// TIA Portal project "P10" (V20)

(* hardware
DEVICE "S7-1200 station_1"  S7-1200 Station
   slot 0: "Rack_0"  S7-1200 Rack  Rack  V1.0
   slot 1: "PLC_1"  CPU 1214C DC/DC/DC  6ES7 214-1AG40-0XB0  V4.7
*)

// ===== PLC "PLC_1"  CPU 1214C DC/DC/DC =====

VAR_GLOBAL   // PLC tag table "Default tag table"
   "IN" AT %M0.0 : Bool;
   "O_TP" AT %M0.1 : Bool;
   "To_TP" AT %MD2 : Time;
   "To_TON" AT %MD6 : Time;
   "O_TON" AT %M0.2 : Bool;
   "To_TOF" AT %MD10 : Time;
   "O_TOF" AT %M0.3 : Bool;
   "Reset" AT %M0.5 : Bool;
   "To_TONR" AT %MD14 : Time;
   "O_TONR" AT %M0.4 : Bool;
   "OCOUNT_CTU" AT %MW18 : Int;
   "Q_CTU" AT %M0.6 : Bool;
   "cargar" AT %M0.7 : Bool;
   "OCOUNT_CTD" AT %MW20 : Int;
   "Q_CTD" AT %M1.0 : Bool;
   "Incremento" AT %M1.1 : Bool;
   "Decremento" AT %M1.2 : Bool;
   "QD_CTUD_Menor0" AT %M1.3 : Bool;
   "conteo" AT %MW22 : Int;
   "QU_CTUD_MAYOR_PV" AT %M1.4 : Bool;
   "enclavamiento" AT %M2.0 : Bool;
   "Verde" AT %Q0.0 : Bool;
   "Tag_3" AT %MD18 : Time;
   "parada" AT %I0.1 : Bool;
   "Amarillo" AT %Q0.1 : Bool;
   "Rojo" AT %Q0.2 : Bool;
   "5srojo" AT %M2.5 : Bool;
   "Tag_2" AT %I0.2 : Bool;
   "Tag_4" AT %M2.2 : Bool;
   "Contador" AT %M2.3 : Bool;
   "reset_cont_sem" AT %M2.4 : Bool;
END_VAR

// folder: System blocks/Program resources

DATA_BLOCK "IEC_Timer_0_DB_5"   // DB8
{ S7_Optimized_Access := 'TRUE' }
AUTHOR : Simatic
FAMILY : IEC
NAME : IEC_TMR
VERSION : 1.0
// stored: InstanceOfName IEC_TIMER
"IEC_TIMER"
BEGIN
END_DATA_BLOCK

DATA_BLOCK "IEC_Timer_0_DB_4"   // DB9
{ S7_Optimized_Access := 'TRUE' }
AUTHOR : Simatic
FAMILY : IEC
NAME : IEC_TMR
VERSION : 1.0
// stored: InstanceOfName IEC_TIMER
"IEC_TIMER"
BEGIN
END_DATA_BLOCK

DATA_BLOCK "IEC_Timer_0_DB_6"   // DB10
{ S7_Optimized_Access := 'TRUE' }
AUTHOR : Simatic
FAMILY : IEC
NAME : IEC_TMR
VERSION : 1.0
// stored: InstanceOfName IEC_TIMER
"IEC_TIMER"
BEGIN
END_DATA_BLOCK

DATA_BLOCK "IEC_Counter_0_DB_3"   // DB11
{ S7_Optimized_Access := 'TRUE' }
AUTHOR : Simatic
FAMILY : IEC
NAME : CNTR
VERSION : 1.0
// stored: InstanceOfName IEC_COUNTER
"IEC_COUNTER"
BEGIN
END_DATA_BLOCK

// folder: (top level)

ORGANIZATION_BLOCK "Main"   // OB1, LAD, ProgramCycle
TITLE = "Main Program Sweep (Cycle)"
{ S7_Optimized_Access := 'TRUE' }
VERSION : 0.1
   VAR_INPUT
      Initial_Call : Bool;   // Initial call of this OB
      Remanence : Bool;   // =True, if remanent data are available
   END_VAR
BEGIN

REGION Network 1
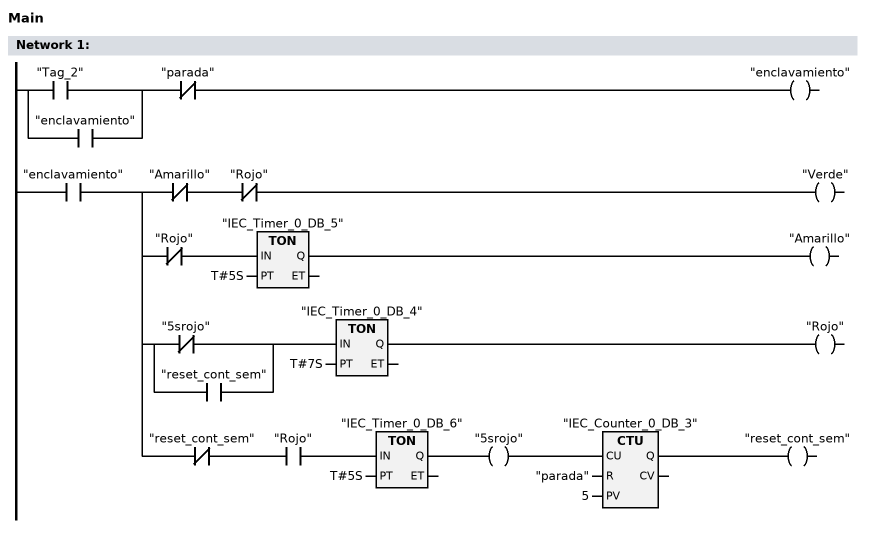
   "enclavamiento" := ("Tag_2" OR "enclavamiento") AND NOT "parada";
   "Verde" := "enclavamiento" AND NOT "Amarillo" AND NOT "Rojo";
   "IEC_Timer_0_DB_5".TON(IN := "enclavamiento" AND NOT "Rojo", PT := T#5S);
   "Amarillo" := "IEC_Timer_0_DB_5".Q;
   "IEC_Timer_0_DB_4".TON(IN := "enclavamiento" AND (NOT "5srojo" OR "reset_cont_sem"), PT := T#7S);
   "Rojo" := "IEC_Timer_0_DB_4".Q;
   "IEC_Timer_0_DB_6".TON(IN := "enclavamiento" AND NOT "reset_cont_sem" AND "Rojo", PT := T#5S);
   "5srojo" := "IEC_Timer_0_DB_6".Q;
   "IEC_Counter_0_DB_3".CTU(CU := "IEC_Timer_0_DB_6".Q, R := "parada", PV := 5);
   "reset_cont_sem" := "IEC_Counter_0_DB_3".Q;
END_REGION
END_ORGANIZATION_BLOCK